{attribute 'linkalways'} 
{attribute 'no_explicit_call' := 'This FB is a CLASS and must be accessed using methods or properties'}
{attribute 'enable_dynamic_creation'}
FUNCTION_BLOCK SetPositionCommand EXTENDS AxisCommand
VAR
	_position : LREAL;
	_mode : SetPositionMode;
END_VAR

METHOD FB_init : BOOL
VAR_INPUT
	bInitRetains : BOOL; // if TRUE, the retain variables are initialized (warm start / cold start)
	bInCopyCode : BOOL;  // if TRUE, the instance afterwards gets moved into the copy code (online change)
	axis : I_Axis;
	position : LREAL;
	mode : SetPositionMode;
END_VAR
_axis := axis;
_position := position;
_mode := mode;
END_METHOD

METHOD PROTECTED  WhileBusy
VAR_INPUT
	CommandState : I_CommandBusyState;
END_VAR
VAR_INST
	_fb : MC_SetPosition;
END_VAR
_fb(
	Axis := _axis._InternalAxisRef,
	Execute := TRUE,
	Position := _position,
	Mode := (_mode = SetPositionMode.Relative)
);

IF _fb.Busy THEN
	RETURN;
END_IF

_fb(Axis := _axis._InternalAxisRef, Execute := FALSE);

IF _fb.Error THEN
	CommandState.SetError(_fb.ErrorID);
	RETURN;
END_IF

CommandState.SetDone();
END_METHOD

END_FUNCTION_BLOCK

(* stored: Version 1.1.0.1, ProductVersion 3.1.4024.12
   POU SetPositionCommand: Id {4cdb3db2-5511-4618-b19e-e8c99b999c4f}, SpecialFunc None
   Folder Constructor: Id {b7dd30ac-bab1-44d9-a58f-2d5e6daac3d0}
   Method FB_init: Id {73cd683d-e018-4190-beed-2e076e3f972c}
   Method WhileBusy: Id {3ec3d9d2-53d5-410d-bbee-fb8ae959523c} *)
